PROGRAM PRG_TEST
VAR
	fb_Vector3 : FB_Vector3_Test;
	fb_RMatrix : FB_RMatrix_Test;
END_VAR

TcUnit.RUN();

END_PROGRAM

(* stored: Version 1.1.0.1, ProductVersion 3.1.4024.9
   POU PRG_TEST: Id {5322b863-4755-4304-b115-246eb156f0a8}, SpecialFunc None *)
